FUNCTION_BLOCK QueryServiceHTTP (* Query for Services using HTTP *)
  (* Standard: 61499-2; Description: Copyright (c) 2018 fortiss GmbH This program and the accompanying materials are made available under the terms of the Eclipse Public License 2.0 which is available at https://www.eclipse.org/legal/epl-2.0/ SPDX-License-Identifier: EPL-2.0 *)
  (* Version 1.0, 2018-09-21, Jose Cabral, fortiss GmbH *)
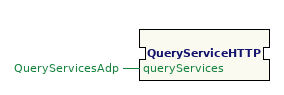
  SOCKETS
    queryServices : QueryServicesAdp;
  END_SOCKETS
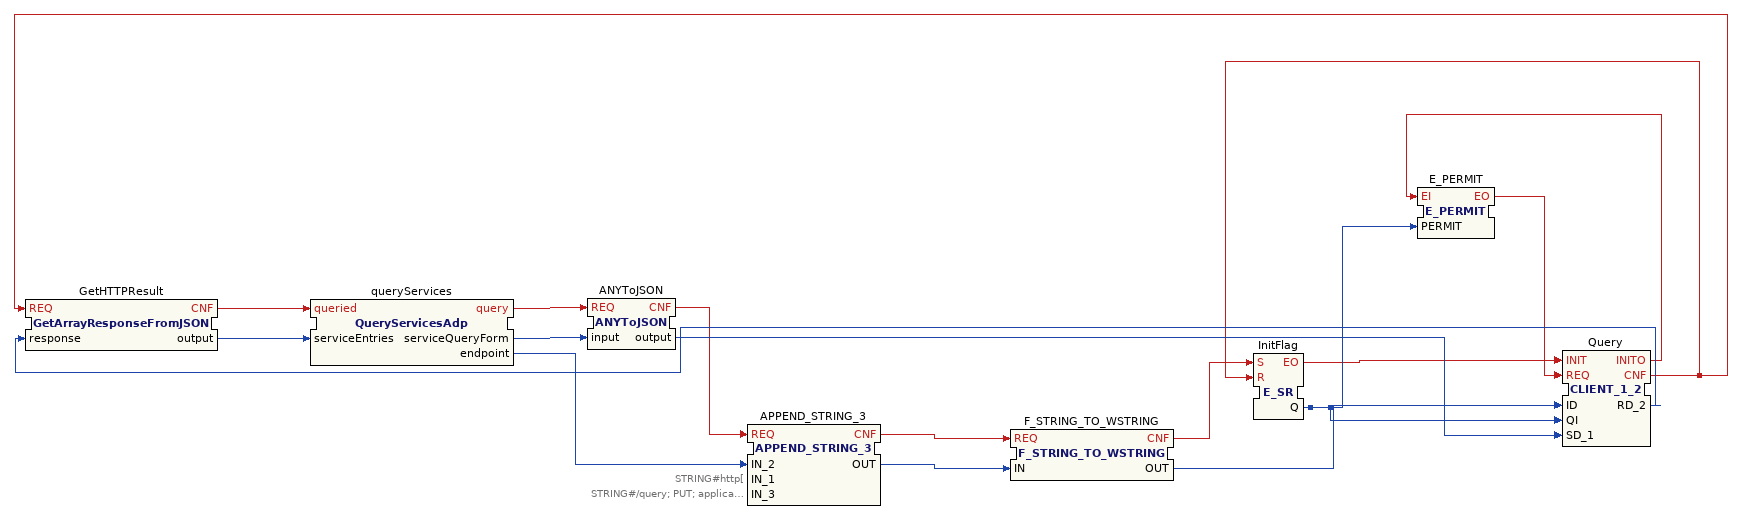
  FBS
    APPEND_STRING_3 : APPEND_STRING_3(IN_1 := STRING#http[, IN_3 := STRING#/query; PUT; application/json]);
    Query : CLIENT_1_2;
    F_STRING_TO_WSTRING : F_STRING_TO_WSTRING;
    InitFlag : E_SR;
    E_PERMIT : E_PERMIT;
    ANYToJSON : ANYToJSON;
    GetHTTPResult : GetArrayResponseFromJSON;
  END_FBS
  EVENT_CONNECTIONS
    APPEND_STRING_3.CNF TO F_STRING_TO_WSTRING.REQ;
    F_STRING_TO_WSTRING.CNF TO InitFlag.S;
    InitFlag.EO TO Query.INIT;
    Query.INITO TO E_PERMIT.EI;
    E_PERMIT.EO TO Query.REQ;
    Query.CNF TO InitFlag.R;
    ANYToJSON.CNF TO APPEND_STRING_3.REQ;
    queryServices.query TO ANYToJSON.REQ;
    Query.CNF TO GetHTTPResult.REQ;
    GetHTTPResult.CNF TO queryServices.queried;
  END_CONNECTIONS
  DATA_CONNECTIONS
    APPEND_STRING_3.OUT TO F_STRING_TO_WSTRING.IN;
    F_STRING_TO_WSTRING.OUT TO Query.ID;
    InitFlag.Q TO E_PERMIT.PERMIT;
    InitFlag.Q TO Query.QI;
    ANYToJSON.output TO Query.SD_1;
    queryServices.serviceQueryForm TO ANYToJSON.input;
    queryServices.endpoint TO APPEND_STRING_3.IN_2;
    Query.RD_2 TO GetHTTPResult.response;
    GetHTTPResult.output TO queryServices.serviceEntries;
  END_CONNECTIONS
END_FUNCTION_BLOCK
